Staubli VAL3: ActionItem.dtx

public num nDistance
public num nMoveId
public num nTimeId
public num nPointId
public InstrItem iInstr[3]
  [0]
    string sType
    string sData
  [1]
    string sType
    string sData
  [2]
    string sType
    string sData
public string sIdTraj
